SUBAPPLICATION AuxInput_Klappen_heben (* Subapplication Type *)
  (* Standard: 61499-2 *)
  (* Version 1.0, 2023-02-11, franz *)
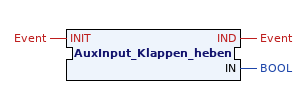
  EVENT_INPUT
    INIT;
  END_EVENT
  EVENT_OUTPUT
    IND;
  END_EVENT
  VAR_OUTPUT
    IN : BOOL;
  END_VAR
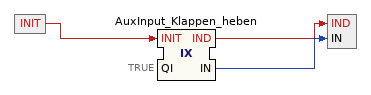
  FBS
    AuxInput_Klappen_heben : IX(QI := TRUE);
  END_FBS
  EVENT_CONNECTIONS
    INIT TO AuxInput_Klappen_heben.INIT;
    AuxInput_Klappen_heben.IND TO IND;
  END_CONNECTIONS
  DATA_CONNECTIONS
    AuxInput_Klappen_heben.IN TO IN;
  END_CONNECTIONS
END_SUBAPPLICATION
